// TIA Portal project "3-Way Smart Sorting Line" (V16)
// Vorlageprojekt für das Buch mit Zielsystem S7-1200

(* hardware
DEVICE "S7-1200-Station_1"  S7-1200 Station
   slot 0: "Baugruppenträger_0"  Rack  V1.0
   slot 1: "PLC_1"  CPU 1211C DC/DC/DC  6ES7 211-1AE40-0XB0  V4.1
*)

// ===== PLC "PLC_1"  CPU 1211C DC/DC/DC =====

VAR_GLOBAL   // PLC tag table "Standard-Variablentabelle"
   "start" AT %I0.0 : Bool;
   "stop" AT %I0.1 : Bool;
   "low" AT %I0.2 : Bool;
   "mid" AT %I0.3 : Bool;
   "high" AT %I0.4 : Bool;
   "main sens" AT %I0.5 : Bool;
   "box detect" AT %I0.6 : Bool;
   "turn table" AT %I0.7 : Bool;
   "left first" AT %I1.0 : Bool;
   "left last" AT %I1.1 : Bool;
   "forward first" AT %I1.2 : Bool;
   "forward last" AT %I1.3 : Bool;
   "right first" AT %I1.4 : Bool;
   "right last" AT %I1.5 : Bool;
   "main con" AT %Q0.0 : Bool;
   "roll +" AT %Q0.2 : Bool;
   "roll -" AT %Q0.3 : Bool;
   "left conv" AT %Q0.4 : Bool;
   "right con" AT %Q0.5 : Bool;
   "forward con" AT %Q0.6 : Bool;
   "box type" AT %MD10 : DInt;
   "Tag_1" AT %M100.5 : Bool;
   "Tag_2" AT %M100.6 : Bool;
   "Tag_3" AT %M101.6 : Bool;
   "Tag_4" AT %M101.3 : Bool;
   "total box" AT %MD14 : DInt;
   "LARGE RATIO" AT %MD18 : Real;
   "alarm" AT %Q0.7 : Bool;
   "reset" AT %I1.6 : Bool;
   "turn +" AT %Q1.0 : Bool;
   "turn-" AT %Q1.1 : Bool;
   "turn 0" AT %I1.7 : Bool;
   "emitter" AT %Q1.2 : Bool;
   "Tag_5" AT %M111.7 : Bool;
END_VAR

// folder: System blocks/Program resources

DATA_BLOCK "IEC_Counter_0_DB"   // DB1
{ S7_Optimized_Access := 'TRUE' }
AUTHOR : Simatic
FAMILY : IEC
NAME : CNTR
VERSION : 1.0
// stored: InstanceOfName IEC_COUNTER
"IEC_COUNTER"
BEGIN
END_DATA_BLOCK

DATA_BLOCK "IEC_Counter_0_DB_1"   // DB2
{ S7_Optimized_Access := 'TRUE' }
AUTHOR : Simatic
FAMILY : IEC
NAME : CNTR
VERSION : 1.0
// stored: InstanceOfName IEC_COUNTER
"IEC_COUNTER"
BEGIN
END_DATA_BLOCK

DATA_BLOCK "IEC_Counter_0_DB_2"   // DB3
{ S7_Optimized_Access := 'TRUE' }
AUTHOR : Simatic
FAMILY : IEC
NAME : CNTR
VERSION : 1.0
// stored: InstanceOfName IEC_COUNTER
"IEC_COUNTER"
BEGIN
END_DATA_BLOCK

// folder: (top level)

FUNCTION "MHJ-PLC-Lab-Function-S71200" : Void   // FC9000, SCL
{ S7_Optimized_Access := 'TRUE' }
VERSION : 0.1
   VAR_TEMP
      rdTimeReturn : Int;
      outputTime : DTL;
      SyncVal : Byte;
      forVal : Int;
      forVal_2 : Int;
      Value : Byte;
   END_VAR
   VAR CONSTANT
      CompVal : Byte := 16#34;
      Value_01 : Byte := 16#11;
      Value_01_DW : DWord := 16#A165_D992;
      Value_02_DW : DWord := 16#58BE_4401;
   END_VAR
BEGIN

   #Value:=PEEK(area := 16#82,
        dbNumber := 0,
        byteOffset := 511);
   #Value := #Value + 1;

   POKE(area := 16#82,
        dbNumber := 0,
        byteOffset := 511,
        value := #Value);

   POKE(area:=16#81,
        dbNumber:=0,
        byteOffset:=1016,
        value:=#Value_01_DW);
   POKE(area := 16#81,
        dbNumber := 0,
        byteOffset := 1020,
        value := #Value_02_DW);

   POKE(area := 16#81,
        dbNumber := 0,
        byteOffset := 511,
        value := B#16#00);

   FOR #forVal := 0 TO 120 DO
       FOR #forVal_2:=0 TO 10 DO
           #rdTimeReturn:=RD_SYS_T(#outputTime);
           #rdTimeReturn := WR_SYS_T(#outputTime);
           #rdTimeReturn := RD_SYS_T(#outputTime);
           #rdTimeReturn := WR_SYS_T(#outputTime);
       END_FOR;
       #SyncVal:= PEEK(area := 16#81,
                      dbNumber := 0,
                      byteOffset := 511);
       IF #SyncVal = #CompVal THEN
          GOTO M_1;
       END_IF;
   END_FOR;
   RETURN;

   M_1:
   POKE(area := 16#81,
        dbNumber := 0,
        byteOffset := 511,
        value := B#16#0);
END_FUNCTION

ORGANIZATION_BLOCK "Main"   // OB1, LAD, ProgramCycle
TITLE = "Main Program Sweep (Cycle)"
{ S7_Optimized_Access := 'TRUE' }
VERSION : 0.1
   VAR_INPUT
      Initial_Call : Bool;   // Initial call of this OB
      Remanence : Bool;   // =True, if remanent data are available
   END_VAR
   VAR_TEMP   // added for the SCL form of the ladder/FBD networks
      _w1 : Bool;
      _w2 : Bool;
      _w3 : Bool;
   END_VAR
BEGIN

REGION Network 1
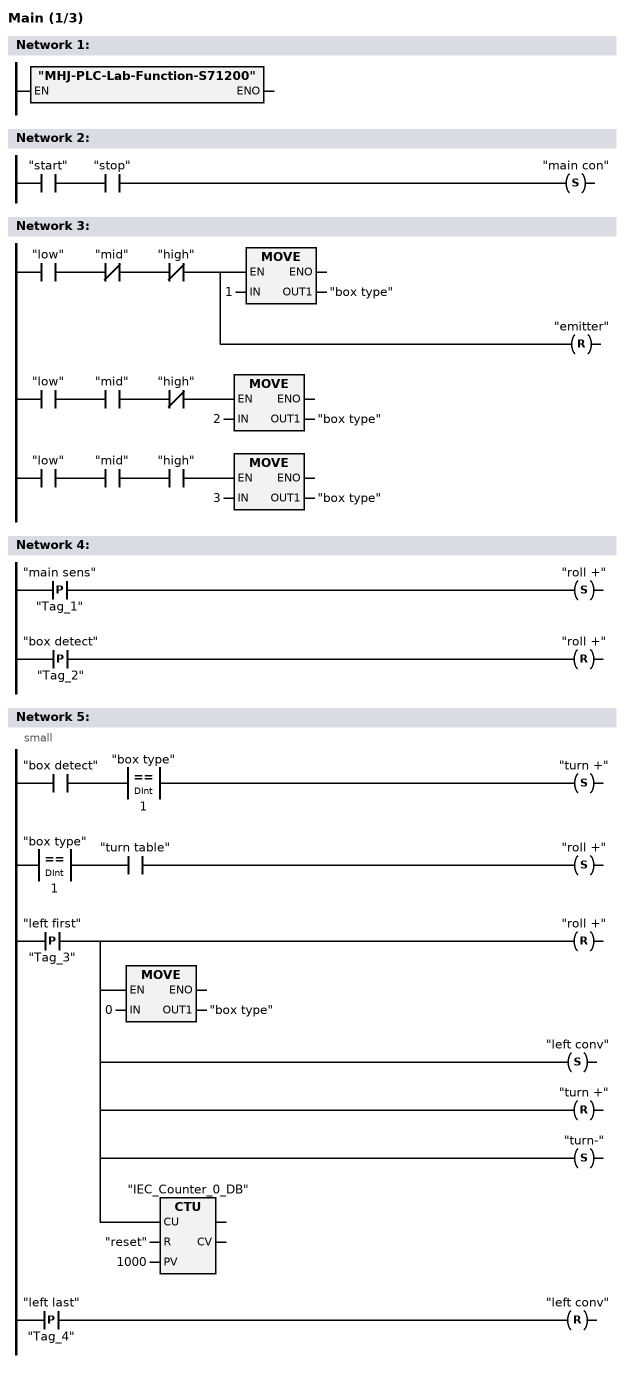
   RUNG wire#powerrail
      "MHJ-PLC-Lab-Function-S71200"()
   END_RUNG
   // the same network as SCL:
   "MHJ-PLC-Lab-Function-S71200"();
END_REGION

REGION Network 2
   RUNG wire#powerrail
      Contact( "start" )
      Contact( "stop" )
      S_Coil( "main con" )
   END_RUNG
   // the same network as SCL:
   IF "start" AND "stop" THEN "main con" := TRUE; END_IF;
END_REGION

REGION Network 3
   RUNG wire#powerrail
      Contact( "low" )
      I_Contact( "mid" )
      I_Contact( "high" )
      wire#w1
      Move(in := 1, out1 => "box type")
   END_RUNG
   RUNG wire#w1
      R_Coil( "emitter" )
   END_RUNG
   RUNG wire#powerrail
      Contact( "low" )
      Contact( "mid" )
      I_Contact( "high" )
      Move(in := 2, out1 => "box type")
   END_RUNG
   RUNG wire#powerrail
      Contact( "low" )
      Contact( "mid" )
      Contact( "high" )
      Move(in := 3, out1 => "box type")
   END_RUNG
   // the same network as SCL:
   IF "low" AND NOT "mid" AND NOT "high" THEN
       "box type" := 1;
       "emitter" := FALSE;
   END_IF;
   IF "low" AND "mid" AND NOT "high" THEN "box type" := 2; END_IF;
   IF "low" AND "mid" AND "high" THEN "box type" := 3; END_IF;
END_REGION

REGION Network 4
   RUNG wire#powerrail
      P_Contact(operand := "main sens", bit := "Tag_1")
      S_Coil( "roll +" )
   END_RUNG
   RUNG wire#powerrail
      P_Contact(operand := "box detect", bit := "Tag_2")
      R_Coil( "roll +" )
   END_RUNG
   // the same network as SCL:
   #_w1 := "main sens" AND NOT "Tag_1";   // rising edge of "main sens"
   "Tag_1" := "main sens";
   IF #_w1 THEN "roll +" := TRUE; END_IF;
   #_w2 := "box detect" AND NOT "Tag_2";   // rising edge of "box detect"
   "Tag_2" := "box detect";
   IF #_w2 THEN "roll +" := FALSE; END_IF;
END_REGION

REGION Network 5
   // small
   IF "box detect" AND ("box type" = 1) THEN "turn +" := TRUE; END_IF;
   IF ("box type" = 1) AND "turn table" THEN "roll +" := TRUE; END_IF;
   #_w1 := "left first" AND NOT "Tag_3";   // rising edge of "left first"
   "Tag_3" := "left first";
   IF #_w1 THEN
       "roll +" := FALSE;
       "box type" := 0;
       "left conv" := TRUE;
       "turn +" := FALSE;
       "turn-" := TRUE;
   END_IF;
   "IEC_Counter_0_DB".CTU(CU := #_w1, R := "reset", PV := 1000);
   #_w2 := "left last" AND NOT "Tag_4";   // rising edge of "left last"
   "Tag_4" := "left last";
   IF #_w2 THEN "left conv" := FALSE; END_IF;
END_REGION

REGION Network 6
   // mid
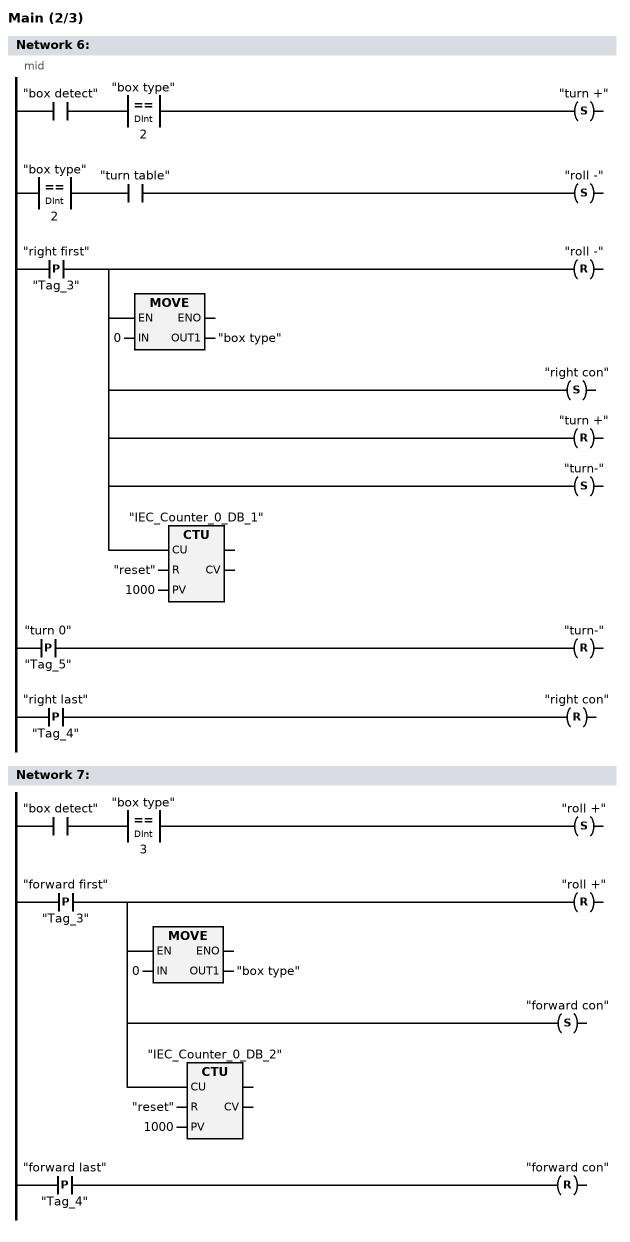
   IF "box detect" AND ("box type" = 2) THEN "turn +" := TRUE; END_IF;
   IF ("box type" = 2) AND "turn table" THEN "roll -" := TRUE; END_IF;
   #_w1 := "right first" AND NOT "Tag_3";   // rising edge of "right first"
   "Tag_3" := "right first";
   IF #_w1 THEN
       "roll -" := FALSE;
       "box type" := 0;
       "right con" := TRUE;
       "turn +" := FALSE;
       "turn-" := TRUE;
   END_IF;
   "IEC_Counter_0_DB_1".CTU(CU := #_w1, R := "reset", PV := 1000);
   #_w2 := "turn 0" AND NOT "Tag_5";   // rising edge of "turn 0"
   "Tag_5" := "turn 0";
   IF #_w2 THEN "turn-" := FALSE; END_IF;
   #_w3 := "right last" AND NOT "Tag_4";   // rising edge of "right last"
   "Tag_4" := "right last";
   IF #_w3 THEN "right con" := FALSE; END_IF;
END_REGION

REGION Network 7
   IF "box detect" AND ("box type" = 3) THEN "roll +" := TRUE; END_IF;
   #_w1 := "forward first" AND NOT "Tag_3";   // rising edge of "forward first"
   "Tag_3" := "forward first";
   IF #_w1 THEN
       "roll +" := FALSE;
       "box type" := 0;
       "forward con" := TRUE;
   END_IF;
   "IEC_Counter_0_DB_2".CTU(CU := #_w1, R := "reset", PV := 1000);
   #_w2 := "forward last" AND NOT "Tag_4";   // rising edge of "forward last"
   "Tag_4" := "forward last";
   IF #_w2 THEN "forward con" := FALSE; END_IF;
END_REGION

REGION Network 8
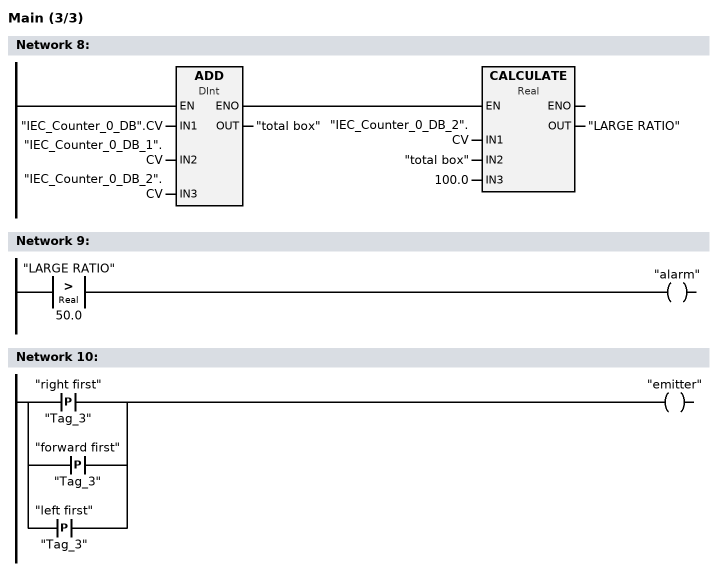
   RUNG wire#powerrail
      { S7_Templates := "SrcType := DInt" } Add(in1 := "IEC_Counter_0_DB".CV, in2 := "IEC_Counter_0_DB_1".CV, in3 := "IEC_Counter_0_DB_2".CV, out => "total box")
      { S7_Templates := "SrcType := Real"; S7_Expression := "(IN1/IN2)*IN3" } Calculate(in1 := "IEC_Counter_0_DB_2".CV, in2 := "total box", in3 := 100.0, out => "LARGE RATIO")
   END_RUNG
   // the same network as SCL:
   "total box" := "IEC_Counter_0_DB".CV + "IEC_Counter_0_DB_1".CV + "IEC_Counter_0_DB_2".CV;
   "LARGE RATIO" := ("IEC_Counter_0_DB_2".CV/"total box")*100.0;
END_REGION

REGION Network 9
   RUNG wire#powerrail
      { S7_Templates := "SrcType := Real" } GT_Contact(in1 := "LARGE RATIO", in2 := 50.0)
      Coil( "alarm" )
   END_RUNG
   // the same network as SCL:
   "alarm" := "LARGE RATIO" > 50.0;
END_REGION

REGION Network 10
   RUNG wire#powerrail
      P_Contact(operand := "right first", bit := "Tag_3")
      wire#w1
      Coil( "emitter" )
   END_RUNG
   RUNG wire#powerrail
      P_Contact(operand := "forward first", bit := "Tag_3")
   END_RUNG wire#w1
   RUNG wire#powerrail
      P_Contact(operand := "left first", bit := "Tag_3")
   END_RUNG wire#w1
   // the same network as SCL:
   #_w1 := "right first" AND NOT "Tag_3";   // rising edge of "right first"
   "Tag_3" := "right first";
   #_w2 := "forward first" AND NOT "Tag_3";   // rising edge of "forward first"
   "Tag_3" := "forward first";
   #_w3 := "left first" AND NOT "Tag_3";   // rising edge of "left first"
   "Tag_3" := "left first";
   "emitter" := #_w1 OR #_w2 OR #_w3;
END_REGION
END_ORGANIZATION_BLOCK